Fanuc KAREL source: NC0002.KL

-- PROVISIONAL review KL for V770-1; original PC SHA256 63932697417cf8d3be0e36b25e77519bb5cab7bfb39f1a41d3e40ee2cfe4958b
-- Incomplete behavior may be omitted. Consult companion uncertainty JSON. Do not deploy.
PROGRAM NC0002
%NOLOCKGROUP
-- UNRESOLVED_LOCAL_POOL 1 cells at code offset 3; source declarations unknown
-- DIRECT_LOCAL_WORD_ACCESS alone does not prove INTEGER, REAL, or BOOLEAN
BEGIN
  -- UNRESOLVED_PC offsets 0-8; opcodes 2B,2C,7B
  -- UNRESOLVED_PC offsets 13-20; opcodes 9D,23
  -- UNRESOLVED_PC offsets 25-38; opcodes 21,9D,57,79
  -- UNRESOLVED_PC offsets 43-57; opcodes 21,9D,52,23
  -- UNRESOLVED_PC offsets 62-67; opcodes 7A
  -- UNRESOLVED_PC offsets 72-90; opcodes 21,2E,52,23
  -- UNRESOLVED_PC offsets 100-104; opcodes 7F
  -- UNRESOLVED_PC offsets 109-113; opcodes 27,AA
  -- UNRESOLVED_PC offsets 118-122; opcodes 7F
END NC0002
